(* Logix 5000 project; controller APM_HW2 Emulate 5570 rev 30.12; software revision 30.00 *)

TASK MainTask (continuous, watchdog 500 ms) : MainProgram

MODULES
   Local : Emulate 5570 (ICP 2, rev 30.12)
      I_O : vendor 1 type 0 code 15 (ICP 3, rev 1.1, Output RPI 150 ms)
END_MODULES

VAR_GLOBAL   (* controller tags *)
   CFull : DINT;
   CON1 : ALIAS FOR Local:3:O.Data[0].2;
   CON2 : ALIAS FOR Local:3:O.Data[0].4;
   LIFT1 : ALIAS FOR Local:3:O.Data[0].1;
   LIFT2 : ALIAS FOR Local:3:O.Data[0].4;
   MC1 : ALIAS FOR Local:3:O.Data[0].3;
   PRESS : ALIAS FOR Local:3:O.Data[0].0;
   START_CONVEYOR1 : BOOL;
   START_CONVEYOR2 : BOOL;
   START_LIFT1 : BOOL;
   START_LIFT2 : BOOL;
   START_MC1 : BOOL;
   START_MC2 : BOOL;
   START_PRESS : BOOL;
   StartS : ALIAS FOR Local:3:I.Data[1].2;
   STOP_CONVEYOR1 : BOOL;
   STOP_CONVEYOR2 : BOOL;
   Stop_I : ALIAS FOR Local:3:I.Data[1].7;
   STOP_LIFT1 : BOOL;
   STOP_LIFT2 : BOOL;
   STOP_MC1 : BOOL;
   STOP_PRESS : BOOL;
   TCON_1 : TIMER := (PRE := 1200);   // Timer Conveyor 1 process
   TCON_2 : TIMER := (PRE := 2000);
   TLIFT_1 : TIMER := (PRE := 500);
   TLIFT_2 : TIMER := (PRE := 2500);
   TMC1 : TIMER := (PRE := 1500);
   TPRESS : TIMER := (PRE := 3500);
END_VAR

PROGRAM MainProgram   (* main routine MainRoutine *)
VAR
   Action_000 : SFC_ACTION := (Status := 16#0020_0000, PauseTimer := 1);
   Action_001 : SFC_ACTION := (Status := 16#0020_0000, PauseTimer := 1);
   Action_002 : SFC_ACTION := (Status := 16#0020_0000, PauseTimer := 1);
   Action_003 : SFC_ACTION := (Status := 16#0020_0000, PauseTimer := 1);
   Action_004 : SFC_ACTION := (Status := 16#0020_0000, PauseTimer := 1);
   Action_005 : SFC_ACTION := (Status := 16#0020_0000, PauseTimer := 1);
   Action_006 : SFC_ACTION := (Status := 16#0020_0000, PauseTimer := 1);
   Action_007 : SFC_ACTION := (Status := 16#0020_0000, PauseTimer := 1);
   Action_008 : SFC_ACTION := (Status := 16#0020_0000, PauseTimer := 1);
   Action_009 : SFC_ACTION := (Status := 16#0020_0000, PauseTimer := 1);
   Action_010 : SFC_ACTION := (Status := 16#0020_0000, PauseTimer := 1);
   Action_011 : SFC_ACTION := (Status := 16#0020_0000, PauseTimer := 1);
   Action_012 : SFC_ACTION := (Status := 16#0020_0000, PauseTimer := 1);
   Action_013 : SFC_ACTION := (Status := 16#0020_0000, PauseTimer := 1);
   Action_014 : SFC_ACTION := (Status := 16#0020_0000, PauseTimer := 1);
   Action_015 : SFC_ACTION := (Status := 16#0020_0000, PauseTimer := 1);
   Action_016 : SFC_ACTION := (Status := 16#0020_0000, PauseTimer := 1);
   Action_017 : SFC_ACTION := (Status := 16#0020_0000, PauseTimer := 1);
   Action_018 : SFC_ACTION := (Status := 16#0020_0000, PauseTimer := 1);
   Action_019 : SFC_ACTION := (Status := 16#0020_0000, PauseTimer := 1);
   Action_020 : SFC_ACTION := (Status := 16#0020_0000, PauseTimer := 1);
   Action_021 : SFC_ACTION := (Status := 16#0020_0000, PauseTimer := 1);
   Action_022 : SFC_ACTION := (Status := 16#0020_0000, PauseTimer := 1);
   Action_023 : SFC_ACTION := (Status := 16#0020_0000, PauseTimer := 1);
   Action_024 : SFC_ACTION := (Status := 16#0020_0000, PauseTimer := 1);
   Action_025 : SFC_ACTION := (Status := 16#0020_0000, PauseTimer := 1);
   Action_026 : SFC_ACTION := (Status := 16#0020_0000, PauseTimer := 1);
   Action_027 : SFC_ACTION := (Status := 16#0020_0000, PauseTimer := 1);
   Agi_1 : SFC_STEP := (Status := 16#0020_0000, PauseTimer := 1, PRE := 1000);
   Atom_1 : SFC_STEP := (Status := 16#0020_0000, PauseTimer := 1, PRE := 1000);
   Atom_2 : SFC_STEP := (Status := 16#0020_0000, PauseTimer := 1, PRE := 1000);
   CONTENT : BOOL;
   Dec_1 : SFC_STEP := (Status := 16#0020_0000, PauseTimer := 1, PRE := 1000);
   Dec_2 : SFC_STEP := (Status := 16#0020_0000, PauseTimer := 1, PRE := 1000);
   DesFe_E : SFC_STEP := (Status := 16#0020_0000, PauseTimer := 1, PRE := 1000);
   Dos_1 : SFC_STEP := (Status := 16#0020_0000, PauseTimer := 1, PRE := 1000);
   Dos_2 : SFC_STEP := (Status := 16#0020_0000, PauseTimer := 1, PRE := 1000);
   Dry_1 : SFC_STEP := (Status := 16#0020_0000, PauseTimer := 1, PRE := 1000);
   Dry_2 : SFC_STEP := (Status := 16#0020_0000, PauseTimer := 1, PRE := 1000);
   Esm : SFC_STEP := (Status := 16#0020_0000, PauseTimer := 1, PRE := 1000);
   FREADY : BOOL;
   MAIN_ENGINE : ALIAS FOR Local:3:O.Data[0].31;
   Mill_1 : SFC_STEP := (Status := 16#0020_0000, PauseTimer := 1, PRE := 1000);
   Oven_Init : SFC_STEP := (Status := 16#0020_0000, PauseTimer := 1, PRE := 1000);
   Oven_Step : SFC_STEP := (Status := 16#0020_0000, PauseTimer := 1, PRE := 1200);
   Oven_T : DINT;
   PACK : BOOL;
   Pack_1 : SFC_STEP := (Status := 16#0020_0000, PauseTimer := 1, PRE := 1000);
   Pack_2 : SFC_STEP := (Status := 16#0020_0000, PauseTimer := 1, PRE := 1000);
   Pack_3 : SFC_STEP := (Status := 16#0020_0000, PauseTimer := 1, PRE := 1000);
   Pallet : SFC_STEP := (Status := 16#0020_0000, PauseTimer := 1, PRE := 1000);
   PProc1 : SFC_STEP := (Status := 16#0020_0000, PauseTimer := 1, PRE := 1200);
   PProc2 : SFC_STEP := (Status := 16#0020_0000, PauseTimer := 1, PRE := 1200);
   PREP : BOOL;
   Press_1 : SFC_STEP := (Status := 16#0020_0000, PauseTimer := 1, PRE := 1000);
   Press_2 : SFC_STEP := (Status := 16#0020_0000, PauseTimer := 1, PRE := 1000);
   QC : SFC_STEP := (Status := 16#0020_0000, PauseTimer := 1, PRE := 1000);
   SEL : DINT;   // Selector Baldosa
   Set1 : ALIAS FOR Local:3:I.Data[1].4;
   Set2 : ALIAS FOR Local:3:I.Data[1].5;
   Set3 : ALIAS FOR Local:3:I.Data[1].6;
   Stacker : SFC_STEP := (Status := 16#0020_0000, PauseTimer := 1, PRE := 1000);
   Step_000 : SFC_STEP := (Status := 16#0020_0000, PauseTimer := 1, PRE := 1200);
   Step_001 : SFC_STEP := (TMax := 4000);
   Step_002 : SFC_STEP := (TMax := 5000);
   Step_003 : SFC_STEP := (Status := 16#0020_0000, PauseTimer := 1, TMax := 5000);
   Step_004 : SFC_STEP := (Status := 16#0020_0000, PauseTimer := 1, TMax := 5000);
   Step_005 : SFC_STEP := (Status := 16#0020_0000, PauseTimer := 1, TMax := 5000);
   Step_006 : SFC_STEP := (Status := 16#0020_0000, PauseTimer := 1, TMax := 5000);
   Step_007 : SFC_STEP := (Status := 16#0020_0000, PauseTimer := 1, TMax := 5000);
   Step_008 : SFC_STEP := (Status := 16#0020_0000, PauseTimer := 1, TMax := 5000);
   Step_009 : SFC_STEP := (Status := 16#0020_0000, PauseTimer := 1);
   Step_010 : SFC_STEP := (Status := 16#0020_0000, PauseTimer := 1);
   Step_011 : SFC_STEP := (Status := 16#0020_0000, PauseTimer := 1);
   Step_012 : SFC_STEP := (Status := 16#0020_0000, PauseTimer := 1);
   Step_013 : SFC_STEP := (Status := 16#0020_0000, PauseTimer := 1);
   Step_014 : SFC_STEP := (Status := 16#0020_0000, PauseTimer := 1);
   Step_015 : SFC_STEP := (Status := 16#0020_0000, PauseTimer := 1);
   Step_016 : SFC_STEP := (Status := 16#0020_0000, PauseTimer := 1);
   Step_017 : SFC_STEP := (Status := 16#0020_0000, PauseTimer := 1);
   Step_018 : SFC_STEP := (Status := 16#0020_0000, PauseTimer := 1);
   Step_019 : SFC_STEP := (Status := 16#0020_0000, PauseTimer := 1);
   Step_020 : SFC_STEP := (Status := 16#0020_0000, PauseTimer := 1);
   Step_021 : SFC_STEP := (Status := 16#0020_0000, PauseTimer := 1);
   Step_022 : SFC_STEP := (Status := 16#0020_0000, PauseTimer := 1);
   Step_023 : SFC_STEP := (Status := 16#0020_0000, PauseTimer := 1);
   Step_024 : SFC_STEP := (Status := 16#0020_0000, PauseTimer := 1);
   Step_025 : SFC_STEP := (Status := 16#0020_0000, PauseTimer := 1);
   Step_026 : SFC_STEP := (Status := 16#0020_0000, PauseTimer := 1);
   Step_027 : SFC_STEP := (Status := 16#0020_0000, PauseTimer := 1);
   Step_028 : SFC_STEP := (Status := 16#0020_0000, PauseTimer := 1);
   Step_029 : SFC_STEP := (Status := 16#0020_0000, PauseTimer := 1);
   Step_030 : SFC_STEP := (Status := 16#0020_0000, PauseTimer := 1);
   Step_031 : SFC_STEP := (Status := 16#0020_0000, PauseTimer := 1);
   Step_032 : SFC_STEP := (Status := 16#0020_0000, PauseTimer := 1);
   Step_033 : SFC_STEP := (Status := 16#0020_0000, PauseTimer := 1);
   STOP : ALIAS FOR Local:3:I.Data[1].1;
   TAG : BOOL;
   TPRESS_1 : TIMER := (PRE := 1500);
   Tran_000 : BOOL;
   Tran_001 : BOOL;
   Tran_002 : BOOL;
   Tran_003 : BOOL;
   Tran_004 : BOOL;
   Tran_005 : BOOL;
   Tran_006 : BOOL;
   Tran_007 : BOOL;
   Tran_008 : BOOL;
   Tran_009 : BOOL;
   Tran_010 : BOOL;
   Tran_011 : BOOL;
   Tran_012 : BOOL;
   Tran_013 : BOOL;
   Tran_018 : BOOL;
   Tran_019 : BOOL;
   Tran_024 : BOOL;
   Tran_025 : BOOL;
   Tran_030 : BOOL;
   Tran_031 : BOOL;
   Tran_032 : BOOL;
   Tran_033 : BOOL;
   Tran_034 : BOOL;
   Tran_036 : BOOL;
   Tran_037 : BOOL;
   Tran_038 : BOOL;
   Tran_039 : BOOL;
   Tran_040 : BOOL;
   Tran_041 : BOOL;
   Tran_042 : BOOL;
   Trat : SFC_STEP := (Status := 16#0020_0000, PauseTimer := 1, PRE := 1000);
   var_c : DINT;
   Vtam_1 : SFC_STEP := (Status := 16#0020_0000, PauseTimer := 1, PRE := 1000);
   VTam_E : SFC_STEP := (Status := 16#0020_0000, PauseTimer := 1, PRE := 1000);
END_VAR
VAR {public}
   BOTTLER : BOOL;
   Ctask : DINT;
   Esm_PProc : SFC_STEP := (Status := 16#0020_0000, PauseTimer := 1, PRE := 2400);
   IO_1 : BOOL;
   Reset : BOOL;
   Stage : DINT;
   Start : ALIAS FOR Local:3:I.Data[1].0;
   Start_GC : BOOL;
   Start_GC1 : BOOL;
   Stop_DT : BOOL := 1;
   TC_1 : DINT;   // Cuantas Cajas de Baldosas tipo 1 hay terminadas
   TC_2 : DINT;   // Cuantas Cajas de Baldosas tipo 2 hay terminadas
   TC_3 : DINT;   // Cuantas Cajas de Baldosas tipo 3 hay terminadas
   WASHER : BOOL;
END_VAR

ROUTINE MainRoutine   (* ladder *)
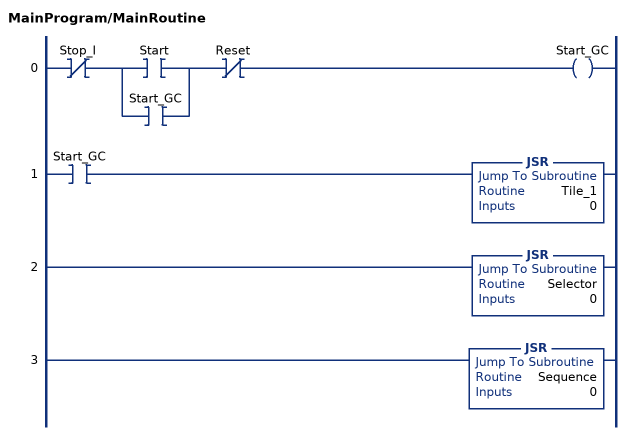
   0: XIO(Stop_I)[XIC(Start) ,XIC(Start_GC) ]XIO(Reset)OTE(Start_GC);
   1: XIC(Start_GC)JSR(Tile_1,0);
   2: JSR(Selector,0);
   3: JSR(Sequence,0);
END_ROUTINE

ROUTINE Selector   (* ladder *)
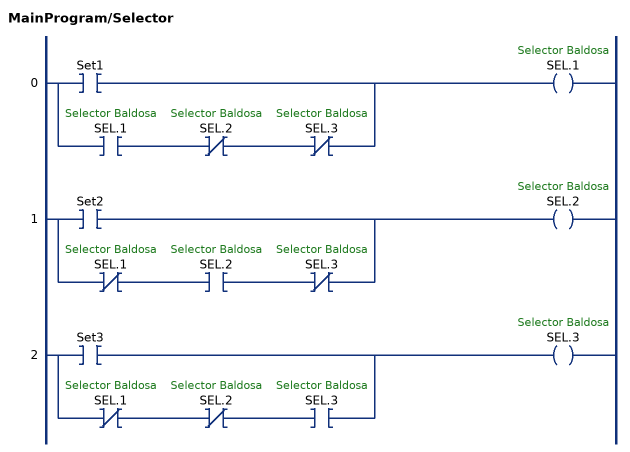
   0: [XIC(Set1) ,XIC(SEL.1) XIO(SEL.2) XIO(SEL.3) ]OTE(SEL.1);
   1: [XIC(Set2) ,XIO(SEL.1) XIC(SEL.2) XIO(SEL.3) ]OTE(SEL.2);
   2: [XIC(Set3) ,XIO(SEL.1) XIO(SEL.2) XIC(SEL.3) ]OTE(SEL.3);
END_ROUTINE

ROUTINE Sequence   (* ladder *)
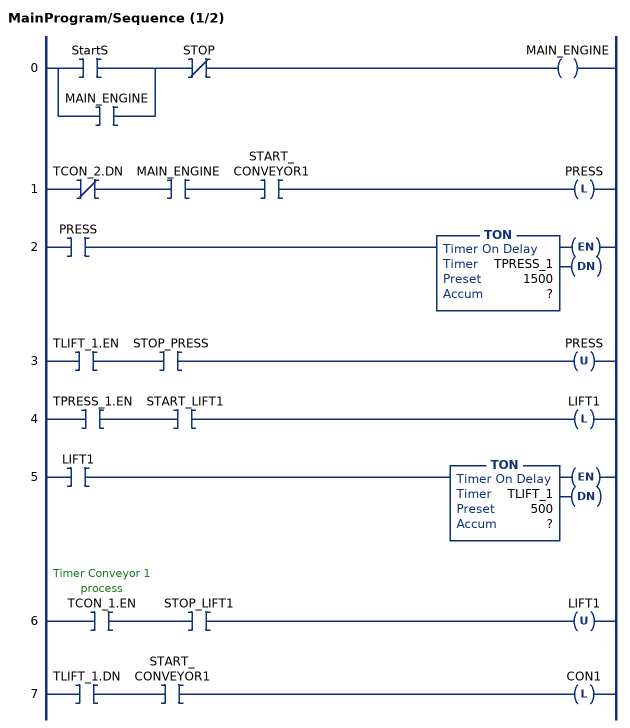
   0: [XIC(StartS) ,XIC(MAIN_ENGINE) ]XIO(STOP)OTE(MAIN_ENGINE);
   1: XIO(TCON_2.DN)XIC(MAIN_ENGINE)XIC(START_CONVEYOR1)OTL(PRESS);
   2: XIC(PRESS)TON(TPRESS_1,?,?);
   3: XIC(TLIFT_1.EN)XIC(STOP_PRESS)OTU(PRESS);
   4: XIC(TPRESS_1.EN)XIC(START_LIFT1)OTL(LIFT1);
   5: XIC(LIFT1)TON(TLIFT_1,?,?);
   6: XIC(TCON_1.EN)XIC(STOP_LIFT1)OTU(LIFT1);
   7: XIC(TLIFT_1.DN)XIC(START_CONVEYOR1)OTL(CON1);
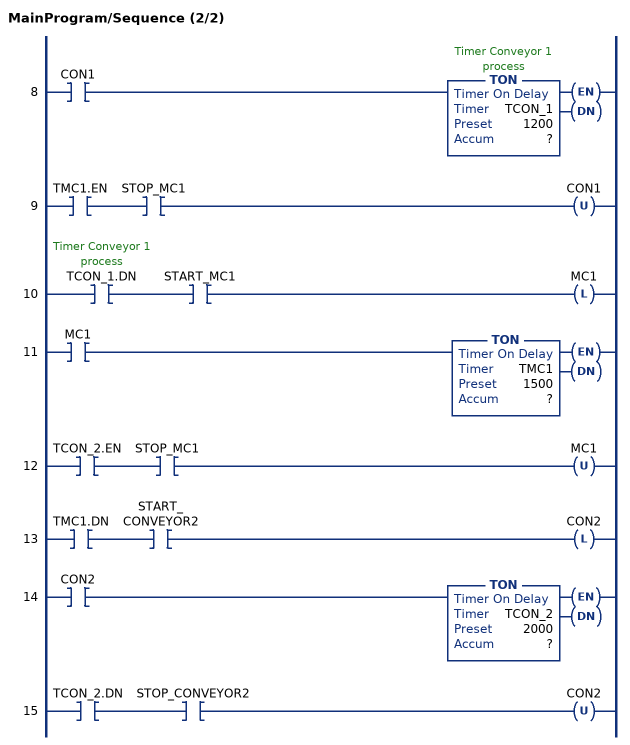
   8: XIC(CON1)TON(TCON_1,?,?);
   9: XIC(TMC1.EN)XIC(STOP_MC1)OTU(CON1);
   10: XIC(TCON_1.DN)XIC(START_MC1)OTL(MC1);
   11: XIC(MC1)TON(TMC1,?,?);
   12: XIC(TCON_2.EN)XIC(STOP_MC1)OTU(MC1);
   13: XIC(TMC1.DN)XIC(START_CONVEYOR2)OTL(CON2);
   14: XIC(CON2)TON(TCON_2,?,?);
   15: XIC(TCON_2.DN)XIC(STOP_CONVEYOR2)OTU(CON2);
END_ROUTINE

ROUTINE Tile_1   (* sequential function chart *)
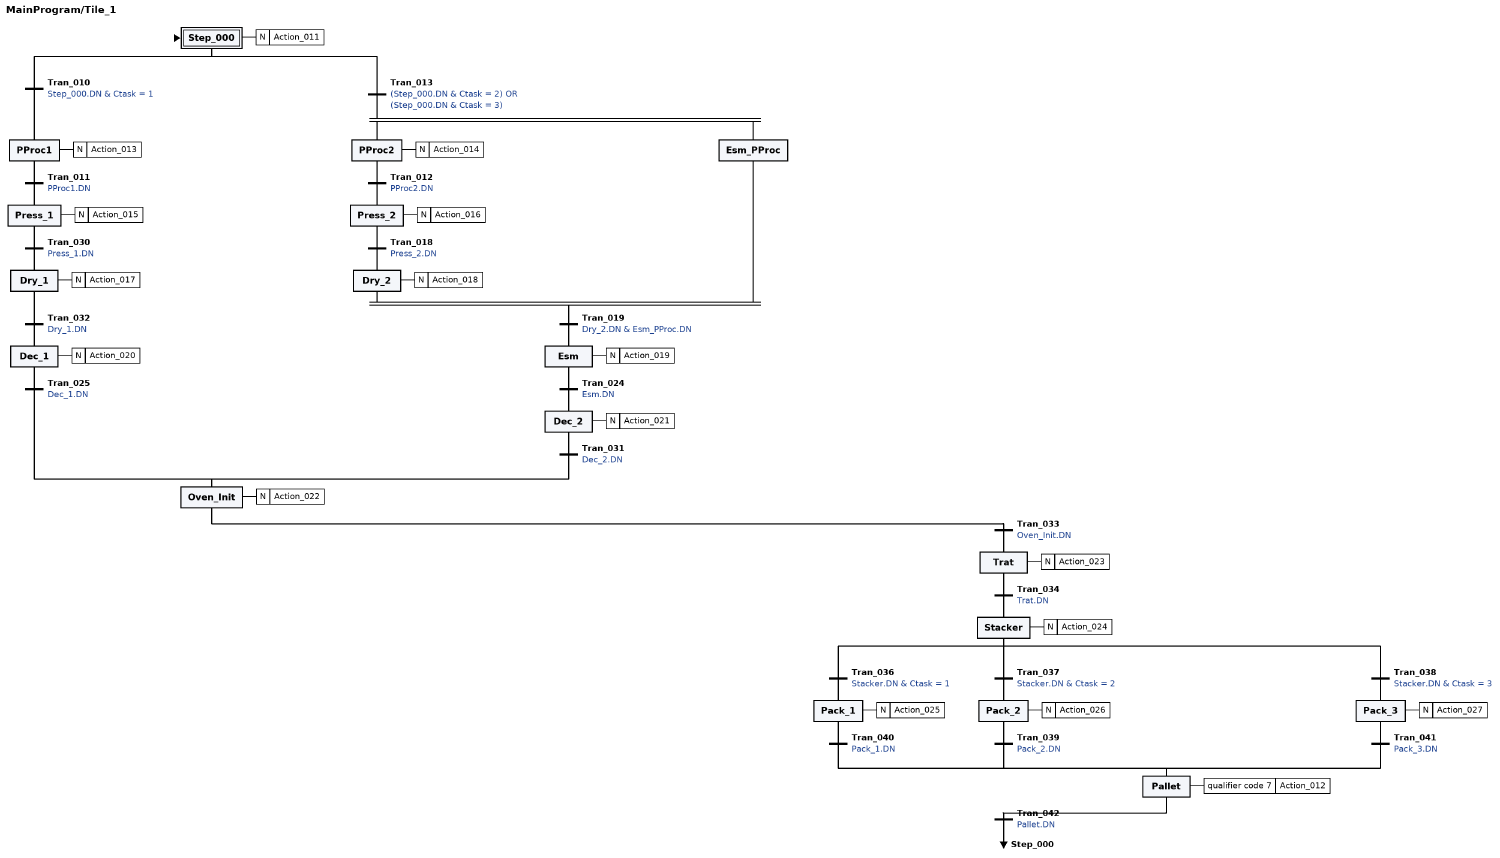
   INITIAL_STEP Step_000:
      ACTION Action_011 (N):
         Stage := 0;
         IF Oven_Init.Count = 0 THEN
         	Oven_T := 5000;
         	TC_1 := 0;
         	TC_2 := 0;
         	TC_3 := 0;
         ELSE
         	Oven_T := 1000;
         END_IF;
         IF SEL = 2 THEN
         	Ctask := 1;
         	ELSIF SEL = 4 THEN
         	Ctask := 2;
         	ELSIF SEL = 8 THEN
         	Ctask := 3;
         END_IF;
      END_ACTION
   END_STEP
   TRANSITION Tran_033 FROM Oven_Init TO Trat
      := Oven_Init.DN
         
   END_TRANSITION
   TRANSITION Tran_013 FROM Step_000 TO (PProc2, Esm_PProc)
      := (Step_000.DN & Ctask = 2) OR (Step_000.DN & Ctask = 3)
   END_TRANSITION
   TRANSITION Tran_010 FROM Step_000 TO PProc1
      := Step_000.DN & Ctask = 1
         
   END_TRANSITION
   STEP Trat:
      ACTION Action_023 (N):
         Stage :=7;
      END_ACTION
   END_STEP
   STEP PProc1:
      ACTION Action_013 (N):
         Stage := 1;
      END_ACTION
   END_STEP
   STEP PProc2:
      ACTION Action_014 (N):
         Stage := 1;
      END_ACTION
   END_STEP
   STEP Esm_PProc:
   END_STEP
   TRANSITION Tran_034 FROM Trat TO Stacker
      := Trat.DN
         
   END_TRANSITION
   TRANSITION Tran_011 FROM PProc1 TO Press_1
      := PProc1.DN
         
   END_TRANSITION
   TRANSITION Tran_012 FROM PProc2 TO Press_2
      := PProc2.DN
         
   END_TRANSITION
   STEP Stacker:
      ACTION Action_024 (N):
         Stage :=8;
         
      END_ACTION
   END_STEP
   STEP Press_1:
      ACTION Action_015 (N):
         Stage := 2;
      END_ACTION
   END_STEP
   STEP Press_2:
      ACTION Action_016 (N):
         Stage := 2;
      END_ACTION
   END_STEP
   TRANSITION Tran_036 FROM Stacker TO Pack_1
      := Stacker.DN & Ctask = 1
         
   END_TRANSITION
   TRANSITION Tran_037 FROM Stacker TO Pack_2
      := Stacker.DN & Ctask = 2
   END_TRANSITION
   TRANSITION Tran_038 FROM Stacker TO Pack_3
      := Stacker.DN & Ctask = 3
   END_TRANSITION
   TRANSITION Tran_030 FROM Press_1 TO Dry_1
      := Press_1.DN
   END_TRANSITION
   TRANSITION Tran_018 FROM Press_2 TO Dry_2
      := Press_2.DN
   END_TRANSITION
   STEP Pack_1:
      ACTION Action_025 (N):
         Stage :=9;
         
         IF (Pack_1.Count MOD 4) = 0 THEN
         	CFull :=1;
         ELSE
         	CFull := 0;
         END_IF;
      END_ACTION
   END_STEP
   STEP Pack_2:
      ACTION Action_026 (N):
         Stage :=9;
         
         IF (Pack_2.Count MOD 4) = 0 THEN
         	CFull :=1;
         ELSE
         	CFull := 0;
         END_IF;
      END_ACTION
   END_STEP
   STEP Pack_3:
      ACTION Action_027 (N):
         Stage :=9;
         
         IF (Pack_3.Count MOD 4) = 0 THEN
         	CFull :=1;
         ELSE
         	CFull := 0;
         END_IF;
      END_ACTION
   END_STEP
   STEP Dry_1:
      ACTION Action_017 (N):
         Stage := 3;
      END_ACTION
   END_STEP
   STEP Dry_2:
      ACTION Action_018 (N):
         Stage := 3;
      END_ACTION
   END_STEP
   TRANSITION Tran_040 FROM Pack_1 TO Pallet
      := Pack_1.DN
   END_TRANSITION
   TRANSITION Tran_039 FROM Pack_2 TO Pallet
      := Pack_2.DN
   END_TRANSITION
   TRANSITION Tran_041 FROM Pack_3 TO Pallet
      := Pack_3.DN
   END_TRANSITION
   TRANSITION Tran_032 FROM Dry_1 TO Dec_1
      := Dry_1.DN
   END_TRANSITION
   TRANSITION Tran_019 FROM (Dry_2, Esm_PProc) TO Esm
      := Dry_2.DN & Esm_PProc.DN
   END_TRANSITION
   STEP Esm:
      ACTION Action_019 (N):
         Stage := 4;
      END_ACTION
   END_STEP
   STEP Pallet:
      ACTION Action_012 (qualifier code 7):
         Stage :=10;
         IF CFull =1 THEN
         
         IF Ctask = 1 THEN
         	TC_1 := TC_1+1;
         	ELSIF Ctask = 2 THEN
         	TC_2 := TC_2+1;
         	ELSIF Ctask = 3 THEN
         	TC_3 := TC_3+1;
         END_IF;
         END_IF;
      END_ACTION
   END_STEP
   TRANSITION Tran_024 FROM Esm TO Dec_2
      := Esm.DN
   END_TRANSITION
   TRANSITION Tran_042 FROM Pallet TO Step_000
      := Pallet.DN
   END_TRANSITION
   STEP Dec_1:
      ACTION Action_020 (N):
         Stage := 5;
      END_ACTION
   END_STEP
   STEP Dec_2:
      ACTION Action_021 (N):
         Stage :=5;
      END_ACTION
   END_STEP
   TRANSITION Tran_025 FROM Dec_1 TO Oven_Init
      := Dec_1.DN
   END_TRANSITION
   TRANSITION Tran_031 FROM Dec_2 TO Oven_Init
      := Dec_2.DN
   END_TRANSITION
   STEP Oven_Init:   {Preset := Oven_T}
      ACTION Action_022 (N):
         Stage := 6;
         
      END_ACTION
   END_STEP
END_ROUTINE
END_PROGRAM
